(*
	Steuerwort 1 (STW1)
	Steuerwort 1 SIEMENS Telegramm 10x
	https://cache.industry.siemens.com/dl/files/665/109770665/att_1023132/v2/109770665_PROFIdrive_Statemachine_DOC_V10_de.pdf
*)
{attribute 'pack_mode' := '1'}
TYPE ST_ProfidriveGSM_Control :
STRUCT
	b0_On 							: BIT; 	//ON/OFF (OFF1)
	b1_CoastStop					: BIT; 	//The axis will not coast stop if this bit is set (OFF2)
	b2_QuickStop					: BIT; 	//The axis will not execute quick stop if this bit is set. Quick stop executes a controlled stop on the axis. (OFF3)
	b3_EnableOperation				: BIT; 	//The axis will enable and execute command if all preconditions are set. If a Wake and Shake procedure has to be executed as part of enabling, the transition to state "S4: Operation Enabled" is delayed until the procedure is finished.
	b4_Reserve						: BIT;	//Reserve
	b5_Reserve						: BIT;	//Reserve
	b6_Reserve						: BIT;	//Reserve
	b7_FaultAcknowledge				: BIT;	//Set this bit to reset faults on the drive.
	b8_Reserve						: BIT;	//Reserve
	b9_Reserve						: BIT;	//Reserve	
	b10_ControlPlc					: BIT;	//When not set, no command is accepted from the PLC.	
	b11_Reserved					: BIT;	//Reserve
	b12_Reserved					: BIT;	//Reserve
	b13_Reserved					: BIT;	//Reserve
	b14_Reserved					: BIT;	//Reserve
	b15_Reserved					: BIT;	//Reserve
END_STRUCT
END_TYPE

(* stored: Version 1.1.0.1, ProductVersion 3.1.4024.12
   DUT ST_ProfidriveGSM_Control: Id {99124a78-f6c2-0c02-2e3b-796aa62109cb} *)
